TYPE Framework :
STRUCT
	ComponentIDRecord	: ComponentIdentifier;	// Component Identifier
	Behavior			: DINT;
	OnScan				: BOOL;
	ResetStart			: BOOL;
	ResetDone			: BOOL;
	FullInitRequired	: BOOL;
	EnableStateTrace	: BOOL;
END_STRUCT
END_TYPE

(* stored: Version 1.1.0.1, ProductVersion 3.1.4024.9
   DUT Framework: Id {0debce16-e9dd-49e5-9595-c1dd4525d6b4} *)
